// TIA Portal V20 export
DATA_BLOCK "ControlNodes"   // DB109
// stored: MemoryReserve 100, Namespace Unit1.Em4
   VAR
      em { ExternalWritable := 'False'} : "LAF_typeEmControlNode";
      cm { ExternalWritable := 'False'} : "Unit1.Em4.typeCmControlNode";
      citiMap : "LER_OEM_Data";
      cutter { ExternalWritable := 'False'} : "Unit1.Em4.typeSequenceControlNode";
   END_VAR
   VAR RETAIN
      cmCompensatorAxisZ { ExternalWritable := 'False'} : "LBC_typeAxisControlNode";
      cmFeedingRollAxisB { ExternalWritable := 'False'} : "LBC_typeAxisControlNode";
      cmElectrodeCutterAxisZ { ExternalWritable := 'False'} : "LBC_typeAxisControlNode";
      cmPositionMovingAxisX { ExternalWritable := 'False'} : "LBC_typeAxis64PosControlNode";
      cmFeederCylinderUpDown { ExternalWritable := 'False'} : "LBC_typeTwoWayActuatorControlNode";
      cmCompensatorSafetyPinIdlePosition { ExternalWritable := 'False'} : "LBC_typeDigitalSignalControlNode";
      cmTabDetectSensor { ExternalWritable := 'False'} : "LBC_typeDigitalSignalControlNode";
      cmTapeDetectSensor { ExternalWritable := 'False'} : "LBC_typeDigitalSignalControlNode";
      cmCutterEpcAnalogInput { ExternalWritable := 'False'} : "LBC_typeAnalogInputControlNode";
      cmCompensatorAxisZ_TorqueCal { ExternalWritable := 'False'} : "LER_typeServoTorqueCalControlNode";
      cmFeedingRollAxisB_TorqueCal { ExternalWritable := 'False'} : "LER_typeServoTorqueCalControlNode";
      cmElectrodeCutterAxisZ_TorqueCal { ExternalWritable := 'False'} : "LER_typeServoTorqueCalControlNode";
      cmPositionMovingAxisX_TorqueCal { ExternalWritable := 'False'} : "LER_typeServoTorqueCalControlNode";
   END_VAR
BEGIN
   // cm.brakeTest.compensator.monitoring.error : Compensator Axis Brake Test Error
   // cm.brakeTest.compensator.monitoring.busy : Compensator Axis Brake Test In progress
   // cm.brakeTest.feedingRoll.monitoring.error : Feeding Roll Axis Brake Test Error
   // cm.brakeTest.feedingRoll.monitoring.busy : Feeding Roll Axis Brake Test In progress
   // cm.brakeTest.cutter.monitoring.error : Cutter Axis Brake Test Error
   // cm.brakeTest.cutter.monitoring.busy : Cutter Axis Brake Test In progress
   // cm.brakeTest.positionMoving.monitoring.error : Position moving Axis Brake Test Error
   // cm.brakeTest.positionMoving.monitoring.busy : Position moving Axis Brake Test In progress
END_DATA_BLOCK
